KUKA KRL data list: cell.dat

&ACCESS RVP
&REL 1
DEFDAT cell
  DECL INT nLocalJobCounter = 0
  DECL REAL rLastCycleTimeSec = 24.6
ENDDAT
